// Mitsubishi GX Works2 project: test1   PLC: Q00J

PROGRAM MAIN
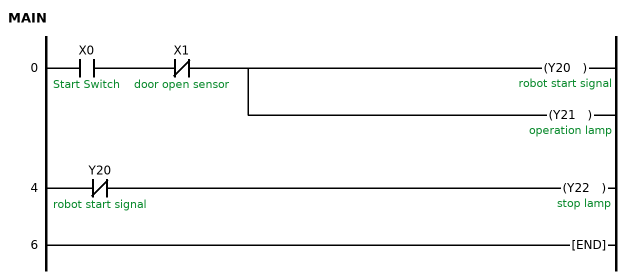
0     LD      X0  ; Start Switch
      ANI     X1  ; door open sensor
      OUT     Y20  ; robot start signal
      OUT     Y21  ; operation lamp
4     LDI     Y20  ; robot start signal
      OUT     Y22  ; stop lamp
6     END
END_PROGRAM
